(* PLC project CHL-DZ-BJDX-11 宁波数字孪生（东方理工）研究院制备薄层色谱全自动化工作站.project, Inovance company InoProShop(V1.9.1.6) InoProShop(V1.9.1.6) *)
(* stored: creationDateTime 2026-06-20T02:01:42.1202334, modificationDateTime 2026-06-18T22:35:27.3049867 *)

FUNCTION_BLOCK FB_Teach
  VAR_IN_OUT
    HMI_Servo : HMI_Servo;
    Servo : servo;
  END_VAR
  VAR
    i : INT;
  END_VAR
  VAR_INPUT
    Mode : INT;
    xEnble : BOOL;
  END_VAR

            IF Mode<>1 AND Servo.bEnabled AND SERVO.bHomed THEN    //没有在自动运行模式下，伺服使能
	//示教点位
	FOR i:=1 TO 10  DO
		IF HMI_Servo.write[i] THEN
		HMI_Servo.position[i]:=Servo.fActPos;
		END_IF
		//运动执行
		IF HMI_Servo.execute[i] THEN
			Servo.fAbsTarget:= HMI_Servo.position[i];
			Servo.xMoveAbs:=TRUE;
		END_IF
		//执行完毕复位
		IF Servo.bAbMoveDone OR Servo.bError  THEN
			Servo.xMoveAbs:=FALSE;
		END_IF
	END_FOR
	
END_IF

          
END_FUNCTION_BLOCK

FUNCTION_BLOCK FB_SERVOAXIS
  VAR_IN_OUT
    AXIS : AXIS_REF_SM3;
  END_VAR
  VAR_INPUT
    xEnable : BOOL;  (* 轴使能 *)
    xHome : BOOL;  (* 回原点命令 *)
    xJogPos : BOOL;  (* 正方向点动 *)
    xJogNeg : BOOL;  (* 负方向点动 *)
    xStop : BOOL;  (* 停止命令 *)
    xMoveAbs : BOOL;  (* 绝对运动启动 *)
    xMoveRel : BOOL;  (* 相对运动启动 *)
    XReset : BOOL;  (* 轴复位 *)
    fAbsTarget : LREAL := 0.0;  (* 绝对位置目标 *)
    fRelTarget : LREAL := 0.0;  (* 相对运动距离 *)
    fVelocity : LREAL := 100.0;  (* 运行速度 *)
    fAcc : LREAL := 1000.0;  (* 加速度 *)
    fDec : LREAL := 1000.0;  (* 减速度 *)
    fJogVel : LREAL := 50.0;  (* 点动速度 *)
  END_VAR
  VAR_OUTPUT
    bEnabled : BOOL;  (* 轴使能状态 *)
    bHomed : BOOL;  (* 原点完成 *)
    bBusy : BOOL;  (* 轴忙状态 *)
    bError : BOOL;  (* 轴报警 *)
    iErrorCode : DINT;  (* 错误代码 *)
    fActPos : LREAL;  (* 实际位置 *)
    fActVel : LREAL;  (* 实际速度 *)
    bAbMoveDone : BOOL;  (* 运动完成 *)
    bReMoveDone : BOOL;  (* 轴使能 *)
  END_VAR
  VAR
    MC_Power : MC_Power;  (* 轴使能 *)
    MC_Home : MC_Home;  (* 回原点 *)
    MC_Homing : MC_Home;  (* 停止 *)
    MC_Halt : MC_Halt;  (* 停止 *)
    MC_MoveAbsolute : MC_MoveAbsolute;  (* 绝对定位 *)
    MC_MoveRelative : MC_MoveRelative;  (* 相对定位 *)
    MC_Jog : MC_Jog;  (* 点动 *)
    MC_Reset : MC_Reset;  (* 轴复位 *)
    bAxisEnabled : BOOL := FALSE;  (* 轴使能标志 *)
    bHomeDone : BOOL := FALSE;  (* 回零完成标志 *)
    bMoving : BOOL := FALSE;  (* 运动中标志 *)
    bHoming : BOOL := FALSE;  (* 回零中标志 *)
  END_VAR

            //轴使能
MC_Power(
	Axis:=AXIS   , 
	Enable:= TRUE  , 
	bRegulatorOn:= xEnable , 
	bDriveStart:=TRUE  , 
	Status=> bEnabled  , 
	bRegulatorRealState=> , 
	bDriveStartRealState=> , 
	Busy=> , 
	Error=>  , 
	ErrorID=>  );
//轴回零
MC_Home(
	Axis:= AXIS, 
	Execute:= xHome , 
	Position:= , 
	Done=> bHomed , 
	Busy=> bHoming , 
	CommandAborted=> , 
	Error=> , 
	ErrorID=> );

//轴复位
MC_Reset(Axis:=AXIS  , 
	Execute:= XReset , 
	Done=> , 
	Busy=> , 
	Error=> ,
	ErrorID=>  );
//轴jog
MC_Jog(
	Axis:=AXIS, 
	JogForward:=xJogPos  , 
	JogBackward:=xJogNeg  , 
	Velocity:=fJogVel  , 
	Acceleration:= fAcc , 
	Deceleration:=fDec  , 
	Jerk:= , 
	Busy=> , 
	CommandAborted=> , 
	Error=> , 
	ErrorId=> );
//轴停止
MC_Halt(
	Axis:=AXIS, 
	Execute:=xStop  , 
	Deceleration:= fDec , 
	Jerk:= , 
	Done=> , 
	Busy=> , 
	CommandAborted=> , 
	Error=> , 
	ErrorID=> );
//轴绝对运动
MC_MoveAbsolute(
	Axis:=AXIS, 
	Execute:= xMoveAbs , 
	Position:= fAbsTarget , 
	Velocity:=fVelocity  , 
	Acceleration:= fAcc , 
	Deceleration:= fDec , 
	Jerk:= , 
	Direction:= , 
	////BufferMode:= , 
	Done=> bAbMoveDone , 
	Busy=> bMoving , 
	////Active=> , 
	CommandAborted=> , 
	Error=> , 
	ErrorID=> );
//轴相对运动
MC_MoveRelative(
	Axis:=AXIS , 
	Execute:=xMoveRel  , 
	Distance:=fRelTarget  , 
	Velocity:= fVelocity , 
	Acceleration:= fAcc , 
	Deceleration:= fDec , 
	Jerk:= , 
	////BufferMode:= , 
	Done=> bReMoveDone, 
	Busy=> , 
	////Active=> , 
	CommandAborted=> , 
	Error=> , 
	ErrorID=> );
	
fActPos:=AXIS.fActPosition ;  //当前位置
fActVel:=AXIS.fActVelocity ;  //当前速度
bError:=MC_Power.Error OR MC_Home.Error OR MC_MoveAbsolute.Error OR MC_MoveAbsolute.Error OR MC_Halt.Error OR MC_Jog.Error OR MC_Reset.Error OR AXIS.nAxisState=1 OR AXIS.nAxisState=2 ;
iErrorCode:=MC_Power.ErrorID OR MC_Home.ErrorID OR MC_MoveAbsolute.ErrorID  OR MC_MoveAbsolute.ErrorID  OR MC_Halt.ErrorID  OR MC_Jog.ErrorId OR MC_Reset.ErrorID  ;





          
END_FUNCTION_BLOCK

FUNCTION_BLOCK FB_cylinder
  VAR_INPUT
    xManualAuto : BOOL := FALSE;  (* 手自动模式：FALSE=手动，TRUE=自动 *)
    xManualExtend : BOOL;  (* 手动伸出 *)
    xManualRetract : BOOL;  (* 手动缩回 *)
    xAutoExtend : BOOL;  (* 自动伸出 *)
    xAutoRetract : BOOL;  (* 自动缩回 *)
    xReset : BOOL;  (* 复位按钮 *)
    xPosExtend : BOOL;  (* 伸出到位传感器 *)
    xPosRetract : BOOL;  (* 缩回到位传感器 *)
    tTimeout : TIME := TIME#5s0ms;  (* 动作超时时间 *)
  END_VAR
  VAR_OUTPUT
    yValve1 : BOOL;  (* 电磁阀1输出：TRUE=伸出，FALSE=缩回 *)
    yValve2 : BOOL;  (* 电磁阀2输出：TRUE=伸出，FALSE=缩回 *)
    bAlarm : BOOL;  (* 报警输出 *)
  END_VAR
  VAR
    bEnableCmd1 : BOOL;  (* 有效的命令1 *)
    bEnableCmd2 : BOOL;  (* 有效的命令1 *)
    tActionTimer : TON;  (* 动作定时器 *)
  END_VAR
  VAR_INPUT
    cylinder_type : INT;  (* 气缸类型 0 单控 1双控 *)
  END_VAR

            

CASE cylinder_type OF
	0:     //单控电池阀
		//命令逻辑选择
		IF xManualAuto  THEN
			//自动模式，使用自动命令
			bEnableCmd1 :=xAutoExtend;
			ELSE
			//手动模式，使用手动命令
			bEnableCmd1 :=xManualExtend  ;
		END_IF
		//控制指令
		IF bEnableCmd1 THEN
			//开始伸出
			yValve1:=TRUE;
			ELSE
			//开始缩回
			yValve1 :=FALSE;
		END_IF
		
	
			tActionTimer(IN := (NOT xPosExtend AND NOT yValve1)  OR   (NOT xPosRetract AND yValve1), PT:=tTimeout );
			bAlarm :=tActionTimer .Q;
	
	1:        //双控电池阀
		//命令逻辑选择
		IF xManualAuto  THEN
			//自动模式，使用自动命令
			bEnableCmd1 :=xAutoExtend;
			bEnableCmd2 :=xAutoRetract;
		ELSE
			//手动模式，使用手动命令
			bEnableCmd1 :=xManualExtend;
			bEnableCmd2 :=xManualRetract;
		END_IF
		//伸出控制指令
		IF bEnableCmd1 THEN
			//开始伸出
			yValve1:=TRUE;
			yValve2:=FALSE;
		ELSE 
			yValve1:=FALSE;
		END_IF
		
		IF bEnableCmd2 THEN
			//开始缩回
			yValve2:=TRUE;
			yValve1:=FALSE;
		ELSE 
			yValve2:=FALSE;
		END_IF
		
			tActionTimer(IN := (NOT xPosExtend AND NOT yValve1)  OR   (NOT xPosRetract AND yValve2), PT:=tTimeout );
			bAlarm :=tActionTimer .Q;
		
END_CASE

IF xReset THEN
	bAlarm:=FALSE ;
END_IF

          
END_FUNCTION_BLOCK

FUNCTION_BLOCK FB_HandWheel
  VAR_IN_OUT
    Axis_Spindle : AXIS_REF_SM3;
    AXIS_1 : AXIS_REF_SM3;
    AXIS_2 : AXIS_REF_SM3;
    AXIS_3 : AXIS_REF_SM3;
    AXIS_4 : AXIS_REF_SM3;
    AXIS_5 : AXIS_REF_SM3;
    AXIS_6 : AXIS_REF_SM3;
    AXIS_7 : AXIS_REF_SM3;
    AXIS_8 : AXIS_REF_SM3;
    AXIS_9 : AXIS_REF_SM3;
  END_VAR
  VAR_INPUT
    Speed_X1 : BOOL;
    Speed_X10 : BOOL;
    Speed_X100 : BOOL;
    Reset : BOOL;
    HandWheel_3Y : BOOL;
    HandWheel_4X : BOOL;
    HandWheel_5Z : BOOL;
    HandWheel_6X : BOOL;
    HandWheel_7Y : BOOL;
    HandWheel_8Y : BOOL;
    HandWheel_9X : BOOL;
    HandWheel_10Z : BOOL;
    HandWheel_11Y : BOOL;
  END_VAR
  VAR
    MC_GearIn_1 : MC_GearIn;
    MC_GearIn_2 : MC_GearIn;
    MC_GearIn_3 : MC_GearIn;
    MC_GearIn_4 : MC_GearIn;
    MC_GearIn_5 : MC_GearIn;
    MC_GearIn_6 : MC_GearIn;
    MC_GearIn_7 : MC_GearIn;
    MC_GearIn_8 : MC_GearIn;
    MC_GearIn_9 : MC_GearIn;
    iDenominator : UDINT;  (* 齿轮比分母 *)
    iMolecule : INT := 1;  (* 齿轮比分子 *)
    MC_GearOut_1 : MC_GearOut;
    TP_0 : TP;
  END_VAR
  VAR_OUTPUT
    xStop_1 : BOOL;
    xStop_2 : BOOL;
    xStop_3 : BOOL;
    xStop_4 : BOOL;
    xStop_5 : BOOL;
    xStop_6 : BOOL;
    xStop_7 : BOOL;
    xStop_8 : BOOL;
    xStop_9 : BOOL;
  END_VAR
  VAR
    R_TRIG_1 : R_TRIG;
    R_TRIG_2 : R_TRIG;
    R_TRIG_3 : R_TRIG;
    R_TRIG_4 : R_TRIG;
    R_TRIG_5 : R_TRIG;
    R_TRIG_6 : R_TRIG;
    R_TRIG_7 : R_TRIG;
    R_TRIG_8 : R_TRIG;
    R_TRIG_9 : R_TRIG;
    R_TRIG_10 : R_TRIG;
    R_TRIG_11 : R_TRIG;
    R_TRIG_12 : R_TRIG;
    R_TRIG_13 : R_TRIG;
    F_TRIG_1 : F_TRIG;
    F_TRIG_2 : F_TRIG;
    F_TRIG_3 : F_TRIG;
    F_TRIG_4 : F_TRIG;
    F_TRIG_5 : F_TRIG;
    F_TRIG_6 : F_TRIG;
    F_TRIG_7 : F_TRIG;
    F_TRIG_8 : F_TRIG;
    F_TRIG_9 : F_TRIG;
  END_VAR
  VAR_OUTPUT
    Error : BOOL;
    ErrorID : WORD;
  END_VAR
  VAR
    MC_GearOut_2 : MC_GearOut;
    MC_GearOut_3 : MC_GearOut;
    MC_GearOut_4 : MC_GearOut;
    MC_GearOut_5 : MC_GearOut;
    MC_GearOut_6 : MC_GearOut;
    MC_GearOut_7 : MC_GearOut;
    MC_GearOut_8 : MC_GearOut;
    MC_GearOut_9 : MC_GearOut;
    newVar : INT;
    newVar1 : INT;
  END_VAR

            //倍率指定
IF Speed_X1  THEN
	iDenominator:=100;
ELSIF Speed_X10 THEN
	iDenominator:=10;
ELSIF Speed_X100 THEN 
    iDenominator:=1;
END_IF
//上升沿检测
R_TRIG_1(CLK:=Speed_X1 );
R_TRIG_2(CLK:=Speed_X10 );
R_TRIG_3(CLK:=Speed_X100 );
R_TRIG_4(CLK:=Reset );
R_TRIG_5(CLK:=HandWheel_3Y  );
R_TRIG_6(CLK:=HandWheel_4X  );
R_TRIG_7(CLK:=HandWheel_5Z );
R_TRIG_8(CLK:=HandWheel_6X );
R_TRIG_9(CLK:=HandWheel_7Y );
R_TRIG_10(CLK:=HandWheel_8Y );
R_TRIG_11(CLK:=HandWheel_9X );
R_TRIG_12(CLK:=HandWheel_10Z );
R_TRIG_13(CLK:=HandWheel_11Y );

//下降沿检测
F_TRIG_1(CLK:=HandWheel_3Y );
F_TRIG_2(CLK:=HandWheel_4X  );
F_TRIG_3(CLK:=HandWheel_5Z );
F_TRIG_4(CLK:=HandWheel_6X );
F_TRIG_5(CLK:=HandWheel_7Y );
F_TRIG_6(CLK:=HandWheel_8Y );
F_TRIG_7(CLK:=HandWheel_9X );
F_TRIG_8(CLK:=HandWheel_10Z );
F_TRIG_9(CLK:=HandWheel_11Y );
//1轴启动啮合
IF R_TRIG_5.Q THEN
	newVar:=newVar+1;
END_IF
IF F_TRIG_1.Q THEN
	newVar1:=newVar1+1;
END_IF

MC_GearIn_1(
	Master:= Axis_Spindle  , 
	Slave:=AXIS_1   , 
	Execute:=R_TRIG_5.Q OR ((R_TRIG_1.Q OR R_TRIG_2.Q OR R_TRIG_3.Q) AND HandWheel_3Y) , 
	RatioNumerator:=iMolecule , 
	RatioDenominator:= iDenominator, 
	Acceleration:= 500, 
	Deceleration:= 800, 
	Jerk:= , 
	//BufferMode:= , 
	InGear=> %MX500.5, 
	Busy=> , 
	//Active=> , 
	CommandAborted=> , 
	Error=> , 
	ErrorID=> );
//2轴启动啮合
MC_GearIn_2(
	Master:= Axis_Spindle, 
	Slave:=AXIS_2 , 
	Execute:=R_TRIG_6.Q OR ((R_TRIG_1.Q OR R_TRIG_2.Q OR R_TRIG_3.Q) AND HandWheel_4X) , 
	RatioNumerator:=iMolecule , 
	RatioDenominator:= iDenominator, 
	Acceleration:= 500, 
	Deceleration:= 800, 
	Jerk:= , 
	//BufferMode:= , 
	InGear=> , 
	Busy=> , 
	//Active=> , 
	CommandAborted=> , 
	Error=> , 
	ErrorID=> );
//3轴启动啮合
MC_GearIn_3(
	Master:= Axis_Spindle, 
	Slave:=AXIS_3 , 
	Execute:= R_TRIG_7.Q OR ((R_TRIG_1.Q OR R_TRIG_2.Q OR R_TRIG_3.Q) AND HandWheel_5Z), 
	RatioNumerator:=iMolecule , 
	RatioDenominator:= iDenominator, 
	Acceleration:= 500, 
	Deceleration:= 800, 
	Jerk:= , 
	//BufferMode:= , 
	InGear=> , 
	Busy=> , 
	//Active=> , 
	CommandAborted=> , 
	Error=> , 
	ErrorID=> );
//4轴启动啮合
MC_GearIn_4(
	Master:= Axis_Spindle, 
	Slave:=AXIS_4 , 
	Execute:=  R_TRIG_8.Q OR ((R_TRIG_1.Q OR R_TRIG_2.Q OR R_TRIG_3.Q) AND HandWheel_6X), 
	RatioNumerator:=iMolecule , 
	RatioDenominator:= iDenominator, 
	Acceleration:= 500, 
	Deceleration:= 800, 
	Jerk:= , 
	//BufferMode:= , 
	InGear=> , 
	Busy=> , 
	//Active=> , 
	CommandAborted=> , 
	Error=> , 
	ErrorID=> );
//5轴启动啮合
MC_GearIn_5(
	Master:= Axis_Spindle, 
	Slave:=AXIS_5 , 
	Execute:= R_TRIG_9.Q OR ((R_TRIG_1.Q OR R_TRIG_2.Q OR R_TRIG_3.Q) AND HandWheel_7Y), 
	RatioNumerator:=iMolecule , 
	RatioDenominator:= iDenominator, 
	Acceleration:= 500, 
	Deceleration:= 800, 
	Jerk:= , 
	//BufferMode:= , 
	InGear=> , 
	Busy=> , 
	//Active=> , 
	CommandAborted=> , 
	Error=> , 
	ErrorID=> );
//6轴启动啮合
MC_GearIn_6(
	Master:= Axis_Spindle, 
	Slave:=AXIS_6 , 
	Execute:= R_TRIG_10.Q OR ((R_TRIG_1.Q OR R_TRIG_2.Q OR R_TRIG_3.Q) AND HandWheel_8Y), 
	RatioNumerator:=iMolecule , 
	RatioDenominator:= iDenominator, 
	Acceleration:= 500, 
	Deceleration:= 800, 
	Jerk:= , 
	//BufferMode:= , 
	InGear=> , 
	Busy=> , 
	//Active=> , 
	CommandAborted=> , 
	Error=> , 
	ErrorID=> );
//7轴启动啮合
MC_GearIn_7(
	Master:= Axis_Spindle, 
	Slave:=AXIS_7 , 
	Execute:= R_TRIG_11.Q OR ((R_TRIG_1.Q OR R_TRIG_2.Q OR R_TRIG_3.Q) AND HandWheel_9X), 
	RatioNumerator:=iMolecule , 
	RatioDenominator:= iDenominator, 
	Acceleration:= 500, 
	Deceleration:= 800, 
	Jerk:= , 
	//BufferMode:= , 
	InGear=> , 
	Busy=> , 
	//Active=> , 
	CommandAborted=> , 
	Error=> , 
	ErrorID=> );
//8轴启动啮合
MC_GearIn_8(
	Master:= Axis_Spindle, 
	Slave:=AXIS_8 , 
	Execute:= R_TRIG_12.Q OR ((R_TRIG_1.Q OR R_TRIG_2.Q OR R_TRIG_3.Q) AND HandWheel_10Z), 
	RatioNumerator:=iMolecule , 
	RatioDenominator:= iDenominator, 
	Acceleration:= 500, 
	Deceleration:= 800, 
	Jerk:= , 
	//BufferMode:= , 
	InGear=> , 
	Busy=> , 
	//Active=> , 
	CommandAborted=> , 
	Error=> , 
	ErrorID=> );
//9轴启动啮合
MC_GearIn_9(
	Master:= Axis_Spindle, 
	Slave:=AXIS_9 , 
	Execute:=  R_TRIG_13.Q OR ((R_TRIG_1.Q OR R_TRIG_2.Q OR R_TRIG_3.Q) AND HandWheel_11Y), 
	RatioNumerator:=iMolecule , 
	RatioDenominator:= iDenominator, 
	Acceleration:= 500, 
	Deceleration:= 800, 
	Jerk:= , 
	//BufferMode:= , 
	InGear=> , 
	Busy=> , 
	//Active=> , 
	CommandAborted=> , 
	Error=> , 
	ErrorID=> );

Error :=MC_GearIn_1.Error OR MC_GearIn_2.Error OR MC_GearIn_3.Error OR MC_GearIn_4.Error OR MC_GearIn_5.Error OR MC_GearIn_6.Error OR MC_GearIn_7.Error OR MC_GearIn_8.Error OR MC_GearIn_9.Error ;  
ErrorID :=MC_GearIn_1.ErrorID OR MC_GearIn_2.ErrorID OR MC_GearIn_3.ErrorID OR MC_GearIn_4.ErrorID OR MC_GearIn_5.ErrorID OR MC_GearIn_6.ErrorID OR MC_GearIn_7.ErrorID OR MC_GearIn_8.ErrorID OR MC_GearIn_9.ErrorID ;  

//1轴断开齿合
MC_GearOut_1(Slave:=AXIS_1 , Execute:= F_TRIG_1.Q AND MC_GearIn_1.InGear , Done=> xStop_1 , Busy=> , Error=> , ErrorID=> );

//2轴断开齿合
MC_GearOut_2(Slave:=AXIS_2 , Execute:= F_TRIG_2.Q AND MC_GearIn_2.InGear , Done=> xStop_2 , Busy=> , Error=> , ErrorID=> );

//3轴断开齿合
MC_GearOut_3(Slave:=AXIS_3 , Execute:= F_TRIG_3.Q AND MC_GearIn_3.InGear , Done=> xStop_3 , Busy=> , Error=> , ErrorID=> );


//4轴断开齿合
MC_GearOut_4(Slave:=AXIS_4 , Execute:= F_TRIG_4.Q AND MC_GearIn_4.InGear , Done=> xStop_4 , Busy=> , Error=> , ErrorID=> );


//5轴断开齿合
MC_GearOut_5(Slave:=AXIS_5 , Execute:= F_TRIG_5.Q AND MC_GearIn_5.InGear , Done=> xStop_5 , Busy=> , Error=> , ErrorID=> );


//6轴断开齿合
MC_GearOut_6(Slave:=AXIS_6 , Execute:= F_TRIG_6.Q AND MC_GearIn_6.InGear , Done=> xStop_6 , Busy=> , Error=> , ErrorID=> );


//7轴断开齿合
MC_GearOut_7(Slave:=AXIS_7 , Execute:= F_TRIG_7.Q AND MC_GearIn_7.InGear , Done=> xStop_7 , Busy=> , Error=> , ErrorID=> );


//8断开齿合
MC_GearOut_8(Slave:=AXIS_8 , Execute:= F_TRIG_8.Q AND MC_GearIn_8.InGear , Done=> xStop_8 , Busy=> , Error=> , ErrorID=> );


//9轴断开齿合
MC_GearOut_9(Slave:=AXIS_9 , Execute:= F_TRIG_9.Q AND MC_GearIn_9.InGear , Done=> xStop_9 , Busy=> , Error=> , ErrorID=> );













          
END_FUNCTION_BLOCK

FUNCTION_BLOCK FB_RB_Control
  VAR_INPUT
    StartCmd : BOOL;
    StopCmd : BOOL;
    PauseCmd : BOOL;
    Reset : BOOL;
    RobotRunning : BOOL;
    RobotStopped : BOOL;
    RobotPaused : BOOL;
    RobotAlarm : BOOL;
    PowerOn : BOOL;
  END_VAR
  VAR_OUTPUT
    StartOut : BOOL;
    StopOut : BOOL;
    PauseOut : BOOL;
    ResetOut : BOOL;
    StatusRun : BOOL;
    StatusStop : BOOL;
    StatusPause : BOOL;
    StatusAlarm : BOOL;
    PowerOnOut : BOOL;
  END_VAR
  VAR
    State : INT := 0;  (* 当前状态 *)
  END_VAR

            (* ================= 报警优先 ================= *)
IF RobotAlarm THEN
    State := 4;
END_IF

CASE State OF

    (* -------- 0：空闲 -------- *)
    0:
        StartOut := FALSE;
        StopOut  := TRUE;
        PauseOut := FALSE;
		ResetOut:=FALSE;
        IF StartCmd AND NOT RobotAlarm THEN
            State := 1;
        END_IF

    (* -------- 1：运行 -------- *)
    1:
		IF NOT PowerOn THEN
			PowerOnOut:=TRUE;
		ELSE
			PowerOnOut:=FALSE;
		END_IF
		IF PowerOn THEN
			StartOut := TRUE;
			StopOut  := FALSE;
			PauseOut := FALSE;
		END_IF
        

        IF StopCmd THEN
            State := 3;
        ELSIF PauseCmd THEN
            State := 2;
        
        END_IF

    (* -------- 2：暂停 -------- *)
    2:
        PauseOut := TRUE;
		StartOut := FALSE ;
        StopOut  := FALSE;
        IF StopCmd THEN
            State := 3;
        ELSIF  StartCmd AND NOT RobotAlarm THEN
            State := 1;
        END_IF

    (* -------- 3：停止 -------- *)
    3:
        StartOut := FALSE;
        StopOut  := TRUE;
        PauseOut := FALSE;

        IF RobotStopped THEN
            State := 0;
        END_IF

    (* -------- 4：报警 -------- *)
    4:
        StartOut := FALSE;
        StopOut  := TRUE;
        PauseOut := FALSE;

        IF  Reset THEN
			ResetOut:=TRUE;
            State := 0;
        END_IF

END_CASE

(* ================= 状态输出 ================= *)
StatusRun   := (State = 1);
StatusPause := (State = 2);
StatusStop  := (State = 0) OR (State = 3);
StatusAlarm := (State = 4);
          
END_FUNCTION_BLOCK

FUNCTION_BLOCK FB_Mode
  VAR_INPUT
    xStart : BOOL;  (* 启动按钮 *)
    xStop : BOOL;  (* 停止按钮 *)
    xReset : BOOL;  (* 复位按钮 *)
    xAutoMode : BOOL;  (* TRUE=自动模式，FALSE=手动模式 *)
    xFault : BOOL;  (* 故障信号 *)
    xEmergency : BOOL;  (* 急停信号（急停按下为FALSE） *)
  END_VAR
  VAR_OUTPUT
    bRed : BOOL;  (* 红灯 *)
    bYellow : BOOL;  (* 黄灯 *)
    bGreen : BOOL;  (* 绿灯 *)
    bBuzzer : BOOL;  (* 蜂鸣器 *)
    iState : INT;  (* 设备状态: 0=停止, 1=运行, 2=故障, 3=急停 *)
    bAuto : BOOL;  (* 自动模式指示 *)
  END_VAR
  VAR
    iDeviceState : INT := 0;  (* 0=停止, 1=运行, 2=故障, 3=急停 *)
    tBuzzerPulse : TON;  (* 蜂鸣器脉冲 *)
    tFlashTimer : TON;  (* 闪烁定时器 *)
    tShortBeep : TON;  (* 短鸣定时器 *)
    tEmergencyBeep : TON;  (* 急停蜂鸣器定时器 *)
    tEmergencyBeep1 : TON;  (* 蜂鸣器激活 *)
    bBuzzerActive : BOOL := FALSE;  (* 蜂鸣器激活 *)
    bFlashFlag : BOOL;  (* 闪烁标志 *)
    bBeepOnce : BOOL := FALSE;  (* 单次蜂鸣标志 *)
    bEmergencyBuzzer : BOOL := FALSE;  (* 急停蜂鸣器标志 *)
    bEmergencyActive : BOOL := FALSE;  (* 急停激活标志 *)
    ALT_0 : ALT;
    ALT_1 : ALT;
    TON_0 : TON;
    ALT_2 : ALT;
    TON_1 : TON;
    TON_2 : TON;
  END_VAR
  VAR_INPUT
    bWarning_alarm : BOOL;
  END_VAR

            // 模式状态
bAuto := xAutoMode;

// 状态机
CASE iDeviceState OF
    EN_功能块状态.停止:  // 停止状态
        IF NOT xEmergency THEN
            iDeviceState := EN_功能块状态.急停;  // 急停
            bEmergencyActive := TRUE;
        ELSIF xFault THEN
            iDeviceState := EN_功能块状态.故障;  // 故障
            bBuzzerActive := TRUE;
        ELSIF (bAuto AND xStart)  THEN
		 bBeepOnce := TRUE;  // 启动短鸣
		  iDeviceState := EN_功能块状态.初始化;  // 初始化

        END_IF;
    
    EN_功能块状态.运行:  // 运行状态
        IF NOT xEmergency THEN
            iDeviceState := EN_功能块状态.急停;  // 急停
            bEmergencyActive := TRUE;
        ELSIF xFault THEN
            iDeviceState := EN_功能块状态.故障;  // 故障
            bBuzzerActive := TRUE;
        ELSIF xStop THEN
            iDeviceState := EN_功能块状态.停止;  // 停止
            bBeepOnce := TRUE;  // 停止短鸣
        END_IF;
        
    EN_功能块状态.故障:  // 故障状态
        IF NOT xEmergency THEN
            iDeviceState := EN_功能块状态.急停;  // 急停
            bEmergencyActive := TRUE;
        ELSIF xReset AND NOT xFault THEN
            iDeviceState := EN_功能块状态.停止;  // 停止
            bBuzzerActive := FALSE;
			bBuzzer:=FALSE;
        END_IF;
        
    EN_功能块状态.急停:  // 急停状态
        // 急停复位需要：急停信号解除 + 复位按钮按下
        IF  xEmergency AND xReset THEN
            iDeviceState := EN_功能块状态.停止;  // 停止
            bEmergencyActive := FALSE;
            bEmergencyBuzzer := FALSE;
			bBuzzer:=FALSE;
        END_IF;
	EN_功能块状态.初始化:  //初始化状态
	 TON_0(IN:=TRUE , PT:=T#3S );
		IF TON_0.Q THEN
		iDeviceState := EN_功能块状态.运行;  // 运行
		END_IF 
END_CASE;

// 急停蜂鸣器控制（急停时蜂鸣器以不同频率鸣响）
IF  bEmergencyActive THEN
    tEmergencyBeep(IN := NOT tEmergencyBeep.Q, PT := T#2S );
	ALT_1(xExecute:= tEmergencyBeep.Q, xOut:=bBuzzer );  // 急停时蜂鸣器响2秒，停2秒	
END_IF;

//三色灯控制
// 闪烁定时器
tFlashTimer(IN := NOT tFlashTimer.Q, PT := T#500MS);
ALT_0(xExecute:=tFlashTimer.Q , xOut:=bFlashFlag );

CASE iDeviceState OF
    EN_功能块状态.停止:  // 停止状态
        IF bAuto THEN
            bYellow := TRUE;           // 自动模式：黄灯常亮
        ELSE
            bYellow := bFlashFlag;     // 手动模式：黄灯闪烁
        END_IF;
		 bGreen :=FALSE;
		 bRed :=FALSE;
        
    EN_功能块状态.运行:  // 运行状态
        bGreen := TRUE;
         bRed :=FALSE;
		  bYellow := FALSE; 
    EN_功能块状态.故障:  // 故障状态
        bRed := TRUE;
         bGreen :=FALSE;
		 bYellow := FALSE; 
    EN_功能块状态.急停:  // 急停状态
        bRed := bFlashFlag;  // 红灯闪烁
		bGreen :=FALSE;
		 bYellow := FALSE; 
END_CASE;
tShortBeep(IN := bBeepOnce AND NOT bEmergencyActive, PT := T#500MS);
// 蜂鸣器控制
IF bBeepOnce AND NOT bEmergencyActive THEN
	bBuzzer := TRUE;  // 短鸣
    IF tShortBeep.Q THEN
        bBeepOnce := FALSE;
       bBuzzer := FALSE;
    END_IF;
    
END_IF;

// 故障时蜂鸣器（非急停状态时生效）
IF NOT bEmergencyActive AND xFault  THEN
    tBuzzerPulse(IN := NOT tBuzzerPulse.Q, PT := T#500MS);
ALT_2(xExecute:= tBuzzerPulse.Q, xOut:= bBuzzer);
END_IF;


//蜂鸣器5S后停止
TON_2(IN:=iDeviceState=2 OR iDeviceState=3 OR bWarning_alarm ,PT:=T#5S);
IF TON_2.Q THEN
	bBuzzer:=FALSE;
END_IF

IF bWarning_alarm AND NOT TON_2.Q THEN
	bBuzzer:=TRUE;
	
END_IF
IF bWarning_alarm  THEN
	 bRed := TRUE;
	  
END_IF

IF xReset THEN
	bBuzzer:=FALSE;
	bRed := FALSE;
END_IF



// 输出状态
iState := iDeviceState;



          
END_FUNCTION_BLOCK
